# EPICS substitutions: multicastTestApp/Db/user.substitutions
# Example substitutions file

file "db/dbExample1.db" {
    { user = "tomytsai" }
}

file db/dbExample2.db {
    pattern { user, no, scan }
        { "tomytsai", 1, "1 second" }
        { "tomytsai", 2, "2 second" }
        { "tomytsai", 3, "5 second" }
}
